(* IEC 61131-3 sources: beckhoffAutomationInterface/ST/Shark, 4 files *)

(* ---- GVL_Shark.st ---- *)
{attribute 'qualified_only'}
VAR_GLOBAL
	nMaxMotorSpeed 	: LREAL 	:= 100.0;	// Global speed limit shared across the project
	sPlantName 		: STRING 	:= 'Shark';	// Human-readable plant/project name
END_VAR

(* ---- FB_Motor.st ---- *)
FUNCTION_BLOCK FB_Motor
VAR_INPUT
	bStart 	: BOOL;				// Start command
END_VAR
VAR_OUTPUT
	eState 		: E_MotorState;		// Current motor state
	stStatus 	: ST_MotorStatus;	// Current motor status
END_VAR
VAR
	fSpeed 	: LREAL := 0;		// Current speed, ramped up while running
END_VAR

// Main cyclic logic of the motor function block
IF bStart THEN
	eState 	:= E_MotorState.Running;
	fSpeed 	:= F_ClampSpeed(fSpeed := fSpeed + 1.0, fMax := 100.0);
ELSE
	eState 	:= E_MotorState.Idle;
	fSpeed 	:= 0;
END_IF

stStatus.bRunning 	:= (eState = E_MotorState.Running);
stStatus.nErrorCode := 0;

METHOD Init : BOOL
VAR_INPUT
END_VAR

// One-time initialization, called once from MAIN on the first cycle
fSpeed 	:= 0;
eState 	:= E_MotorState.Idle;
Init 	:= TRUE;

METHOD Reset : BOOL
VAR_INPUT
END_VAR

// Clears speed, state, and status back to defaults
fSpeed 				:= 0;
eState 				:= E_MotorState.Idle;
stStatus.bRunning 	:= FALSE;
stStatus.nErrorCode := 0;
Reset 				:= TRUE;

(* ---- FB_MotorBase.st ---- *)
{abstract}
FUNCTION_BLOCK FB_MotorBase
VAR
END_VAR

{abstract}
METHOD Stop : BOOL
VAR_INPUT
END_VAR

(* ---- MAIN.st ---- *)
PROGRAM MAIN
VAR
	sHelloWorld 	: STRING 	:= 'Hello, World!'; 	// Sample greeting string
	nCounter		: DINT 		:= 0; 					// Increments once every PLC cycle
	fbMotor			: FB_Motor;							// Motor function block instance
	bInitDone		: BOOL 		:= FALSE;				// Latches once Init() has run
	bResetDone		: BOOL 		:= FALSE;				// Latches the result of the last Reset() call
END_VAR

// Increment the counter on every cycle
nCounter := nCounter + 1;

// Call Init() once on the first cycle
IF NOT bInitDone THEN
	bInitDone := fbMotor.Init();
END_IF

// Periodically reset the motor (demo trigger)
IF nCounter MOD 1000 = 0 THEN
	bResetDone := fbMotor.Reset();
END_IF

// Drive the motor and run its main cyclic logic
fbMotor(bStart := TRUE);
